FUNCTION_BLOCK CSV_WRITER_MEAN (* Writes averaged PV system data to a CSV file. *)
  (* Standard: 61499-2; Description: This function block is intended for field testing purposes only. It should not be used in a real system, since the file size would grow indefinitely. *)
  (* Version 1.0, 2017-09-08, Marc Jakobi, HTW Berlin *)
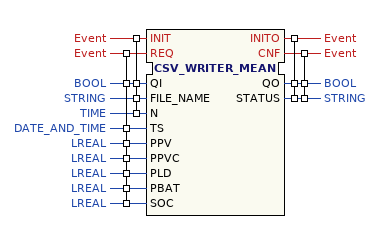
  EVENT_INPUT
    INIT WITH QI, FILE_NAME, N; (* Initialization Request *)
    REQ WITH QI, TS, PPV, PPVC, PLD, PBAT, SOC; (* Normal Execution Request *)
  END_EVENT
  EVENT_OUTPUT
    INITO WITH QO, STATUS; (* Initialization Confirm *)
    CNF WITH QO, STATUS; (* Execution Confirmation *)
  END_EVENT
  VAR_INPUT
    QI : BOOL; (* Input event qualifier *)
    FILE_NAME : STRING := output.csv; (* Output file name *)
    N : TIME := T#1m; (* Averaging interval *)
    TS : DATE_AND_TIME; (* Time stamp *)
    PPV : LREAL; (* Uncurtailed PV power *)
    PPVC : LREAL; (* Curtailed PV power *)
    PLD : LREAL; (* Electric consumption *)
    PBAT : LREAL; (* Battery transfer *)
    SOC : LREAL;
  END_VAR
  VAR_OUTPUT
    QO : BOOL; (* Output event qualifier *)
    STATUS : STRING; (* Service status *)
  END_VAR
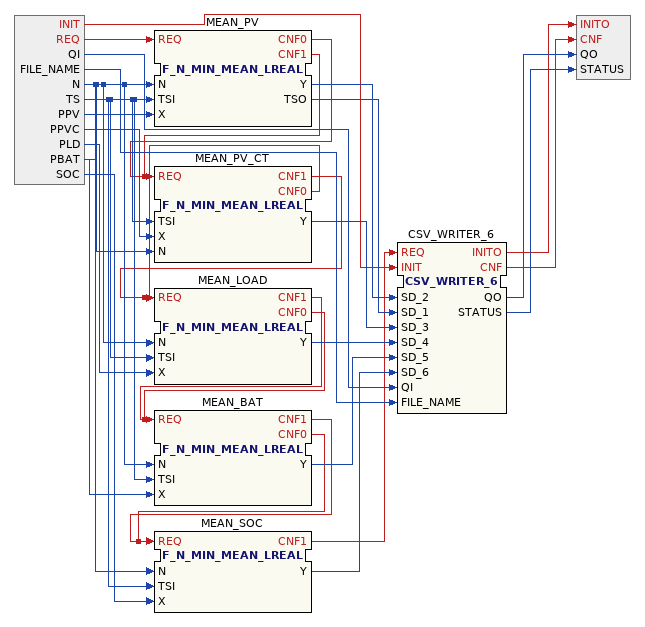
  FBS
    CSV_WRITER_6 : CSV_WRITER_6;
    MEAN_PV : F_N_MIN_MEAN_LREAL;
    MEAN_PV_CT : F_N_MIN_MEAN_LREAL;
    MEAN_LOAD : F_N_MIN_MEAN_LREAL;
    MEAN_BAT : F_N_MIN_MEAN_LREAL;
    MEAN_SOC : F_N_MIN_MEAN_LREAL;
  END_FBS
  EVENT_CONNECTIONS
    REQ TO MEAN_PV.REQ;
    MEAN_PV.CNF0 TO MEAN_PV_CT.REQ;
    MEAN_PV.CNF1 TO MEAN_PV_CT.REQ;
    MEAN_PV_CT.CNF1 TO MEAN_LOAD.REQ;
    MEAN_PV_CT.CNF0 TO MEAN_LOAD.REQ;
    MEAN_LOAD.CNF1 TO MEAN_BAT.REQ;
    MEAN_LOAD.CNF0 TO MEAN_BAT.REQ;
    MEAN_BAT.CNF1 TO MEAN_SOC.REQ;
    MEAN_BAT.CNF0 TO MEAN_SOC.REQ;
    MEAN_SOC.CNF1 TO CSV_WRITER_6.REQ;
    INIT TO CSV_WRITER_6.INIT;
    CSV_WRITER_6.INITO TO INITO;
    CSV_WRITER_6.CNF TO CNF;
  END_CONNECTIONS
  DATA_CONNECTIONS
    N TO MEAN_PV.N;
    TS TO MEAN_PV.TSI;
    PPV TO MEAN_PV.X;
    MEAN_PV.Y TO CSV_WRITER_6.SD_2;
    MEAN_PV.TSO TO CSV_WRITER_6.SD_1;
    MEAN_PV_CT.Y TO CSV_WRITER_6.SD_3;
    TS TO MEAN_PV_CT.TSI;
    PPVC TO MEAN_PV_CT.X;
    N TO MEAN_PV_CT.N;
    N TO MEAN_LOAD.N;
    TS TO MEAN_LOAD.TSI;
    PLD TO MEAN_LOAD.X;
    N TO MEAN_BAT.N;
    TS TO MEAN_BAT.TSI;
    PBAT TO MEAN_BAT.X;
    N TO MEAN_SOC.N;
    TS TO MEAN_SOC.TSI;
    SOC TO MEAN_SOC.X;
    MEAN_LOAD.Y TO CSV_WRITER_6.SD_4;
    MEAN_BAT.Y TO CSV_WRITER_6.SD_5;
    MEAN_SOC.Y TO CSV_WRITER_6.SD_6;
    QI TO CSV_WRITER_6.QI;
    FILE_NAME TO CSV_WRITER_6.FILE_NAME;
    CSV_WRITER_6.QO TO QO;
    CSV_WRITER_6.STATUS TO STATUS;
  END_CONNECTIONS
END_FUNCTION_BLOCK
